// TwinCAT 3 PLC project PLC01
// ProgramVersion: 3.1.4024.0
// libraries:
//   Tc2_Standard, * (Beckhoff Automation GmbH)
//   Tc2_System, * (Beckhoff Automation GmbH)
//   Tc2_Utilities, * (Beckhoff Automation GmbH)
//   Tc3_Module, * (Beckhoff Automation GmbH)
//   VisuDialogs, * (System)
// project tree:
//   DUTs/ st01.TcDUT, st_DirContentInfo.TcDUT
//   / GlobalTextList.TcGTLO, PlcTask.TcTTO, Visualization Manager.TcVMO (not stored), VISU_TASK.TcTTO
//   GVLs/ GVL.TcGVL
//   POUs/ FB_AutoResetBool.TcPOU, FB_FileCopy.TcPOU, MAIN.TcPOU, prgFileHnd.TcPOU, prgFileManipulation.TcPOU
//   VISUs/ Visualization.TcVIS
// real-time tasks:
//   TASK PlcTask: cycle T#10ms, priority 20, ADS port 350
//   TASK VISU_TASK: cycle T#100000us, priority 30, ADS port 351

CONFIGURATION PLC01
    RESOURCE PLC ON TwinCAT3
        TASK PlcTask(INTERVAL := T#10ms, PRIORITY := 20);
        TASK VISU_TASK(INTERVAL := T#100000us, PRIORITY := 30);
        PROGRAM MAIN WITH PlcTask : MAIN;
        PROGRAM VisuElems_Visu_Prg WITH VISU_TASK : VisuElems.Visu_Prg;
    END_RESOURCE
END_CONFIGURATION

// ---- DUTs/st01.TcDUT
TYPE st01 :
STRUCT
	r1:LREAL;
	i1:INT;
	s1:STRING;
	s2:STRING;
	r2:LREAL;
	i2:INT;
END_STRUCT
END_TYPE

// ---- DUTs/st_DirContentInfo.TcDUT
TYPE st_DirContentInfo :
STRUCT
	fileName:T_MaxString;
	dataCriacao:DT;
END_STRUCT
END_TYPE

// ---- GVLs/GVL.TcGVL
{attribute 'qualified_only'}
VAR_GLOBAL
	updateFileList: BOOL;
END_VAR

// ---- POUs/MAIN.TcPOU
PROGRAM MAIN
VAR
	aStructs:ARRAY[1..20] OF st01;
	
END_VAR

prgFileHnd();
prgFileManipulation();

END_PROGRAM

// ---- POUs/prgFileHnd.TcPOU
PROGRAM prgFileHnd
VAR
	bWrite			: BOOL := FALSE;(* Rising edge starts program execution *)
	sNetId			: T_AmsNetId := '';	(* TwinCAT system network address *)
	sFileName		: T_MaxString := 'MyFile';(* CSV destination file path and name *)
	bError			: BOOL;
	nErrId			: UDINT;
	hFile			: UINT		:= 0;(* File handle of the source file *)
	step			: DWORD 	:= 0;

	fbFileOpen	: FB_FileOpen;(* Opens file *)
	fbFileClose	: FB_FileClose;(* Closes file *)
	fbFileWrite	: FB_FileWrite;(* Reads binary data *)	
	trig:R_trig;
	sErr: STRING;
	sMsg: STRING;
	
	//Read
	bRead: BOOL;
	sFileNameRead:T_MaxString;
	bErrorRead:BOOL;
	nErrIdRead:UDINT;
	stepRead:UINT;
	hFileRead:UINT;
	trigRead:R_TRIG;
	
	fbFileOpenRead	: FB_FileOpen;(* Opens file *)
	fbFileCloseRead	: FB_FileClose;(* Closes file *)
	fbFileRead	: FB_FileRead;(* Reads binary data *)
	
	sMsgRead: STRING;
	sErrRead: STRING;
//	sFilePath:T_MaxString:='C:\Relat\';
	sFullfileName: T_MaxString;
END_VAR

trig(CLK:= bWrite);

CASE step OF 
	0:
		IF trig.Q THEN
			step:=10;
			fbFileOpen(bExecute:= FALSE);
			fbFileClose(bExecute:= FALSE);
			fbFileWrite(bExecute:= FALSE);
			sMsg:='Abrindo arquivo';
			sErr:='';
		END_IF
	10:
		sFullfileName:= concat(prgFileManipulation.path, concat(concat('\', sFileName),'.bkp'));
		fbFileOpen(sNetId:=sNetId , sPathName:= sFullfileName, nMode:= FOPEN_MODEWRITE OR FOPEN_MODEBINARY, 
			ePath:= PATH_GENERIC, bExecute:= TRUE, tTimeout:= T#10S, bError => bError, nErrId => nErrId);
		IF NOT fbFileOpen.bBusy THEN
			IF NOT fbFileOpen.bError THEN
				step:=20;
				hFile:= fbFileOpen.hFile;
				sMsg:='Escrevendo arquivo';
			ELSE
				step:=100;
				sErr:='Erro ao abrir o arquivo';
			END_IF
		END_IF
	20:
		fbFileWrite(sNetId:= sNetId, hFile:= hFile,	pWriteBuff:=ADR(main.aStructs), cbWriteLen:= SIZEOF(MAIN.aStructs),
			bExecute:= TRUE,tTimeout:=T#20S, bError => bError, nErrId => nErrId);
		IF NOT fbFileWrite.bBusy THEN
			IF NOT fbFileWrite.bError THEN
				step:=30;
				sMsg:='Arquivo salvo';
			ELSE
				step:=100;
				sErr:='Erro ao escrever o arquivo';	
			END_IF
		END_IF
	30:
		fbFileClose( sNetId := sNetId, hFile := hFile, bExecute := TRUE, bError => bError, nErrId => nErrId);
		IF NOT fbFileClose.bBusy THEN
			step:=100;
			hFile:=0;
			GVL.updateFileList:=TRUE;
		END_IF
	100:
		IF hFile <> 0 THEN
			step:=30;
		ELSE
			step:=0;
			sMsg:='';
		END_IF
END_CASE

trigRead(CLK:= bRead);
CASE stepRead OF
	0:
		IF trigRead.Q THEN
			stepRead:=10;
			fbFileOpenRead(bExecute:= FALSE);
			fbFileCloseRead(bExecute:= FALSE);
			fbFileRead(bExecute:= FALSE);
			sMsgRead:='Abrindo arquivo';
			sErrRead:='';
		END_IF
	10:
		sFileNameRead:= concat(prgFileManipulation.path, concat('\',prgFileManipulation.selectedLocalFile));
		fbFileOpenRead(sNetId:=sNetId , sPathName:= sFileNameRead, nMode:= FOPEN_MODEREAD OR FOPEN_MODEBINARY, 
			ePath:= PATH_GENERIC, bExecute:= TRUE, tTimeout:= T#10S, bError => bErrorRead, nErrId => nErrIdRead);
		IF NOT fbFileOpenRead.bBusy THEN
			IF NOT fbFileOpenRead.bError THEN
				hFileRead:= fbFileOpenRead.hFile;
				stepRead:=20;
			ELSE
				stepRead:=100;	
				sErrRead:='Erro ao abrir arquivo para leitura';
			END_IF
		END_IF
	20:
		fbFileRead(sNetId:=sNetId ,hFile:=hFileRead ,pReadBuff:=ADR(MAIN.aStructs) ,cbReadLen:=SIZEOF(MAIN.aStructs) ,bExecute:=TRUE , 
			tTimeout:= T#30S,bError=> bErrorRead, nErrId=>nErrIdRead);
		IF NOT fbFileRead.bBusy THEN
			IF NOT fbFileRead.bError THEN
				stepRead:=30;
			ELSE
				stepRead:=100;
				sErrRead:='Erro ao ler o arquivo';
			END_IF
		END_IF
	30:
		fbFileCloseRead( sNetId := sNetId, hFile := hFileRead, bExecute := TRUE, bError => bErrorRead, nErrId => nErrIdRead);
		IF NOT fbFileCloseRead.bBusy THEN
			stepRead:=100;
			hFileRead:=0;
			GVL.updateFileList:=TRUE;
		END_IF
	100:
		IF hFileRead <> 0 THEN
			stepRead:=30;
		ELSE
			stepRead:=0;
			sMsgRead:='';
		END_IF
END_CASE

END_PROGRAM

// ---- POUs/prgFileManipulation.TcPOU
PROGRAM prgFileManipulation
VAR
	//Local
	findFiles:FB_EnumFindFileList;
	path: T_MaxString := 'C:\Relat';
	filesFound:ARRAY[1..iNumFiles] OF ST_FindFileEntry;
	filesInfo:ARRAY[1..iNumFiles] OF st_DirContentInfo;
	nNumFiles: UDINT;
	bFindFiles: BOOL;
	bErr: BOOL;
	nErr: UDINT;
	i: UINT;
	i2: UINT;
	searchPath: T_MaxString;
	findFilesFinished:F_TRIG;
	deleteLocalFile: BOOL;

	
	//USB
	findFilesUSB:FB_EnumFindFileList;
	pathUSB: T_MaxString := 'D:';
	filesFoundUSB:ARRAY[1..iNumFiles] OF ST_FindFileEntry;
	filesInfoUSB:ARRAY[1..iNumFiles] OF st_DirContentInfo;
	nNumFilesUSB: UDINT;
	bFindFilesUSB: BOOL;
	bErrUSB: BOOL;
	nErrUSB: UDINT;
	iUSB: UINT;
	i2USB: UINT;
	searchPathUSB: T_MaxString;
	findFilesFinishedUSB:F_TRIG;
	deleteUSBFile: BOOL;

	
	//File copy
	
	fileCopy:FB_FileCopy;
	fileDelete:FB_FileDelete;
	selectedLocalFile:T_MaxString;
	selectedUSBFile:T_MaxString;
	selectedRowLocal:INT;
	selectedRowUSB:INT;
	copyLocalTOUSB: BOOL;
	copyUSBToLocal: BOOL;

	sFullCopyPathLocal: T_MaxString;
	sFullCopyPathUSB: T_MaxString;
	trigCopyLocalUSB, trigCopyUSBLocal, trigDelLocal, trigDelUSB:R_TRIG;
	copyEndTrig, delEndTrig:F_TRIG;
	sCopyMsg: STRING;
	resetUpdateVar:FB_AutoResetBool;
END_VAR
VAR CONSTANT
	iNumFiles:UINT:=10;
END_VAR

searchPath:= concat(path, '\*.*');
findFiles(
	sNetId:='' , 
	sPathName:= searchPath, 
	eCmd:=, 
	pFindList:= ADR(filesFound), 
	cbFindList:= SIZEOF(filesFound), 
	bExecute:= bFindFiles OR GVL.updateFileList, 
	tTimeout:= T#10S, 
	bBusy=> , 
	bError=> bErr, 
	nErrID=> nErr, 
	bEOE=> , 
	nFindFiles=> nNumFiles);

findFilesFinished(CLK:=findFiles.bBusy);

IF findFilesFinished.Q THEN
	FOR i:= 1 TO iNumFiles DO
		filesInfo[i].fileName:= '';
		filesInfo[i].dataCriacao:= DT#1970-1-1-0:0:0;
	END_FOR
	i:=i2:= 1;

	WHILE i<= iNumFiles AND_THEN filesFound[i].sFileName <> '' DO
		IF filesFound[i].fileAttributes.bArchive THEN
			filesInfo[i2].fileName:= filesFound[i].sFileName;
			filesInfo[i2].dataCriacao:= FILETIME_TO_DT(filesFound[i].creationTime);
			i2:=i2+1;
		END_IF
		i:=i+1;
	END_WHILE
END_IF

//USB
searchPathUSB:= concat(pathUSB, '\*.*');
findFilesUSB(
	sNetId:='' , 
	sPathName:= searchPathUSB, 
	eCmd:=, 
	pFindList:= ADR(filesFoundUSB), 
	cbFindList:= SIZEOF(filesFoundUSB), 
	bExecute:= bFindFilesUSB OR GVL.updateFileList, 
	tTimeout:= T#10S, 
	bBusy=> , 
	bError=> bErrUSB, 
	nErrID=> nErrUSB, 
	bEOE=> , 
	nFindFiles=> nNumFilesUSB);

findFilesFinishedUSB(CLK:=findFilesUSB.bBusy);	

IF findFilesFinishedUSB.Q THEN
	
	FOR i:=1 TO iNumFiles DO
		filesInfoUSB[i].fileName:='';
		filesInfoUSB[i].dataCriacao:= DT#1970-1-1-0:0:0;
	END_FOR
	iUSB:=i2USB:= 1;
    
    WHILE iUSB<= iNumFiles AND_THEN filesFoundUSB[iUSB].sFileName <> '' DO
    	IF filesFoundUSB[iUSB].fileAttributes.bArchive THEN
    		filesInfoUSB[i2USB].fileName:= filesFoundUSB[iUSB].sFileName;
    		filesInfoUSB[i2USB].dataCriacao:= FILETIME_TO_DT(filesFoundUSB[iUSB].creationTime);
    		i2USB:=i2USB+1;
    	END_IF
    	iUSB:=iUSB+1;
    END_WHILE
END_IF

IF selectedRowLocal>= 1 AND selectedRowLocal <= iNumFiles THEN
	selectedLocalFile:=filesInfo[selectedRowLocal].fileName;
END_IF	
IF selectedRowUSB>= 1 AND selectedRowUSB <= iNumFiles THEN
	selectedUSBFile:=filesInfoUSB[selectedRowUSB].fileName;
END_IF	

sFullCopyPathLocal:= concat(path,concat('\',selectedLocalFile));
sFullCopyPathUSB:= concat(pathUSB,concat('\',selectedUSBFile));

trigCopyLocalUSB(CLK:= copyLocalTOUSB);
trigCopyUSBLocal(CLK:= copyUSBToLocal);
trigDelLocal(CLK:= deleteLocalFile);
trigDelUSB(CLK:= deleteUSBFile);

IF trigCopyLocalUSB.Q THEN
	fileCopy.sSrcPathName:=sFullCopyPathLocal;
	fileCopy.sDestPathName:= concat(pathUSB,concat('\',selectedLocalFile));
ELSIF trigCopyUSBLocal.Q THEN
	fileCopy.sSrcPathName:=sFullCopyPathUSB;
	fileCopy.sDestPathName:= concat(path,concat('\',selectedUSBFile));;	
END_IF

fileCopy(
	sSrcNetId:= '', 
	sDestNetId:= '', 
	bExecute:=trigCopyLocalUSB.Q OR trigCopyUSBLocal.Q , 
	tTimeOut:= T#20S, 
	bBusy=> , 
	bError=> , 
	nErrId=> );
	
copyEndTrig(CLK:=fileCopy.bBusy);
IF copyEndTrig.Q THEN
	IF NOT fileCopy.bError THEN
		sCopyMsg:='Arquivo copiado com sucesso';
	ELSE 
		sCopyMsg:= concat('Erro na copia do arquivo : ', UDINT_TO_STRING(fileCopy.nErrId));
	END_IF
	GVL.updateFileList:=TRUE;
END_IF



IF trigDelLocal.Q THEN
	fileDelete.sPathName:= sFullCopyPathLocal;
ELSIF trigDelUSB.Q THEN
	fileDelete.sPathName:= sFullCopyPathUSB;	
END_IF

fileDelete(
	sNetId:= '', 
	sPathName:= , 
	ePath:= , 
	bExecute:= trigDelLocal.Q OR trigDelUSB.Q , 
	tTimeout:= T#20S, 
	bBusy=> , 
	bError=> , 
	nErrId=> );
	
delEndTrig(CLK:= fileDelete.bBusy);
IF delEndTrig.Q THEN
	GVL.updateFileList:=TRUE;
END_IF

//put this on the last line
resetUpdateVar(tResetTime:=T#100MS , bReset:= GVL.updateFileList);

END_PROGRAM

// ---- POUs/FB_FileCopy.TcPOU
FUNCTION_BLOCK FB_FileCopy
VAR_INPUT
	sSrcNetId			: T_AmsNetId;	(* TwinCAT network address of the source file *)
	sSrcPathName		: T_MaxString;	(* Source file path and name *)
	sDestNetId			: T_AmsNetId;	(* TwinCAT network address of the destination file *)
	sDestPathName		: T_MaxString;  (* Destination file path and name *)
	bExecute			: BOOL;			(* Rising edge start fb execution *)
	tTimeOut			: TIME := DEFAULT_ADS_TIMEOUT;(* Max. ADS timeout time *)
END_VAR
VAR_OUTPUT
	bBusy				:BOOL;(* TRUE => File copy execution in progress, FALSE => File copy execution idle *)
	bError				:BOOL;(* TRUE => Error, FALSE => No error *)
	nErrId				:UDINT;(* Error code *)
END_VAR
VAR
	fbFileOpen			:FB_FileOpen;
	fbFileClose			:FB_FileClose;
	fbFileRead			:FB_FileRead;
	fbFileWrite			:FB_FileWrite;

	hSrcFile				:UINT	:= 0;(* File handle of the source file *)
	hDestFile			:UINT	:= 0;(* File handle of the destination file *)

	Step				:DWORD;
	RisingEdge			:R_TRIG;

	buffRead				:ARRAY[1..1000] OF BYTE;(* Buffer *)
	cbReadLength		:UDINT := 0;
END_VAR

RisingEdge(CLK:=bExecute);

CASE Step OF
	0:	(* Idle state *)
		IF RisingEdge.Q THEN
			bBusy := TRUE;
			bError:= FALSE;
			nErrId:=0;
			Step := 1;
			cbReadLength:=0;
			hSrcFile:=0;
			hDestFile:=0;
		END_IF

	1:	(* Open source file *)
		fbFileOpen( bExecute := FALSE );
		fbFileOpen( sNetId := sSrcNetId, sPathName := sSrcPathName,
					nMode := FOPEN_MODEREAD OR FOPEN_MODEBINARY,
					ePath := PATH_GENERIC, tTimeout := tTimeOut, bExecute := TRUE );
		Step := Step + 1;
	2:
		fbFileOpen( bExecute := FALSE );
		IF NOT fbFileOpen.bBusy THEN
			IF fbFileOpen.bError THEN
				nErrId := fbFileOpen.nErrId;
				bError := TRUE;
				Step := 50;
			ELSE
				hSrcFile := fbFileOpen.hFile;
				Step := Step + 1;
			END_IF
		END_IF

	3:	(* Open destination file *)
		fbFileOpen( bExecute := FALSE );
		fbFileOpen( sNetId := sDestNetId, sPathName := sDestPathName,
					nMode := FOPEN_MODEWRITE OR FOPEN_MODEBINARY,
					ePath := PATH_GENERIC, tTimeout := tTimeOut, bExecute := TRUE );
		Step := Step+1;
	4:
		fbFileOpen( bExecute := FALSE );
		IF NOT fbFileOpen.bBusy THEN
			IF fbFileOpen.bError THEN
				nErrId := fbFileOpen.nErrId;
				bError := TRUE;
				Step := 50;
			ELSE
				hDestFile := fbFileOpen.hFile;
				Step := Step + 1;
			END_IF
		END_IF

	5:	(* Read data from source file *)
		cbReadLength := 0;
		fbFileRead( bExecute:= FALSE );
		fbFileRead( sNetId:=sSrcNetId, hFile:=hSrcFile,
					pReadBuff:= ADR(buffRead), cbReadLen:= SIZEOF(buffRead),
					bExecute:=TRUE, tTimeout:=tTimeOut );
		Step := Step + 1;
	6:
		fbFileRead( bExecute:= FALSE );
		IF NOT fbFileRead.bBusy THEN
			IF fbFileRead.bError THEN
				nErrId := fbFileRead.nErrId;
				bError := TRUE;
				Step := 50;
			ELSE
				cbReadLength := fbFileRead.cbRead;
				Step := Step + 1;
			END_IF
		END_IF

	7:	(* Write data to destination file *)
		fbFileWrite( bExecute := FALSE );
		fbFileWrite( sNetId:=sDestNetId, hFile:=hDestFile,
					pWriteBuff:= ADR(buffRead), cbWriteLen:= cbReadLength,
					bExecute:=TRUE, tTimeout:=tTimeOut );
		Step := Step + 1;
	8:
		fbFileWrite( bExecute := FALSE );
		IF NOT fbFileWrite.bBusy THEN
			IF fbFileWrite.bError THEN
				nErrId := fbFileWrite.nErrId;
				bError := TRUE;
				Step := 50;
			ELSE
				IF fbFileRead.bEOF THEN (* Check if the EOF flag ist set *)
					Step := 50;	(* Cleanup: close the destination and source files *)
				ELSE
					Step := 5; (* Repeat reading/writing *)
				END_IF
			END_IF
		END_IF

	30:	(* Close the destination file *)
		fbFileClose( bExecute := FALSE );
		fbFileClose( sNetId:=sDestNetId, hFile:=hDestFile, bExecute:=TRUE, tTimeout:=tTimeOut );
		Step := Step + 1;
	31:
		fbFileClose( bExecute := FALSE );
		IF NOT fbFileClose.bBusy THEN
			IF fbFileClose.bError THEN
				nErrId := fbFileClose.nErrId;
				bError := TRUE;
			END_IF
			Step := 50;
			hDestFile := 0;
		END_IF

	40: (* Close source file *)
		fbFileClose( bExecute := FALSE );
		fbFileClose( sNetId:=sSrcNetId, hFile:=hSrcFile, bExecute:=TRUE, tTimeout:=tTimeOut );
		Step := Step + 1;
	41:
		fbFileClose( bExecute := FALSE );
		IF NOT fbFileClose.bBusy THEN
			IF fbFileClose.bError THEN
				nErrId := fbFileClose.nErrId;
				bError := TRUE;
			END_IF
			Step := 50;
			hSrcFile := 0;
		END_IF

	50: (* Error or ready => Cleanup *)
		IF ( hDestFile <> 0 ) THEN
			Step := 30; (* Close the destination file*)
		ELSIF (hSrcFile <> 0 ) THEN
			Step := 40; (* Close the source file *)
		ELSE
			Step := 0;	(* Ready *)
			bBusy := FALSE;
		END_IF

END_CASE

END_FUNCTION_BLOCK

// ---- POUs/FB_AutoResetBool.TcPOU
FUNCTION_BLOCK FB_AutoResetBool
VAR_INPUT
	tResetTime:TIME:=T#100MS;
END_VAR
VAR_OUTPUT
END_VAR
VAR
	t1:TON;
END_VAR
VAR_IN_OUT
	bReset: BOOL;
END_VAR

t1(IN:=bReset , PT:= tResetTime);
IF t1.Q THEN
	bReset:=FALSE;
END_IF

END_FUNCTION_BLOCK

// ---- GlobalTextList.TcGTLO
TEXTLIST GlobalTextList
  607 = '%s'
  576 = '<<< Copiar'
  915 = 'Arquivos'
  449 = 'Carregar'
  770 = 'Copiar >>>'
  642 = 'Criação'
  294 = 'Delete'
  875 = 'Destino'
  166 = 'i1'
  223 = 'i2'
  765 = 'Local'
  253 = 'Mensagem : %s'
  932 = 'Nome'
  814 = 'Nome arquivo'
  762 = 'Origem'
  370 = 'r1'
  76 = 'r2'
  950 = 'Refresh'
  338 = 's1'
  862 = 's2'
  813 = 'Salvar'
  575 = 'USB'
END_TEXTLIST

// ---- VISUs/Visualization.TcVIS
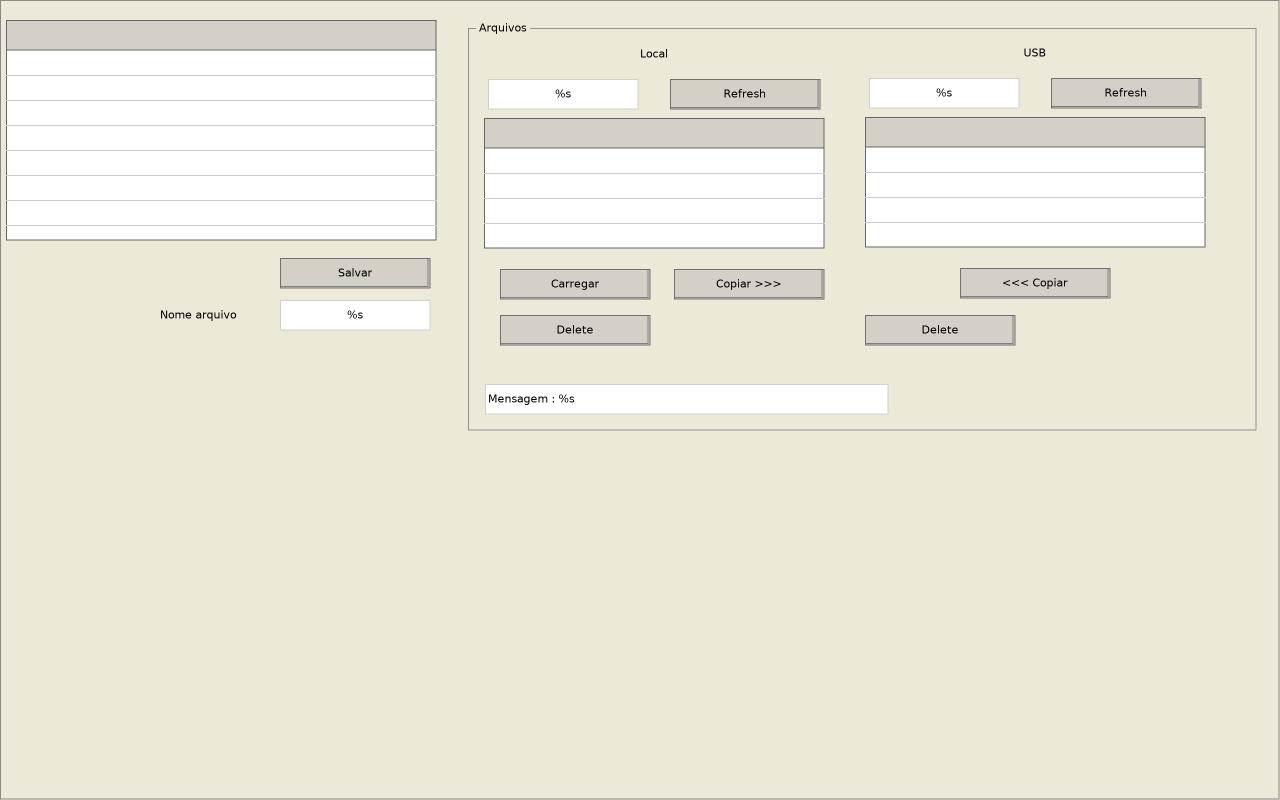
VISUALIZATION Visualization  // 1280x800
    Table (6,20 430x220), data array: MAIN.aStructs
        p3854506369: MAIN.aStructs[INDEX].r1
        p1892666644: MAIN.aStructs[INDEX].i1
        p338671338: MAIN.aStructs[INDEX].s1
        p2170511999: MAIN.aStructs[INDEX].s2
        p3723444502: MAIN.aStructs[INDEX].r2
        p1218418051: MAIN.aStructs[INDEX].i2
    Button (280,258 150x30), "Salvar"
        tap prgFileHnd.bWrite
    Label (144,300 109x30), "Nome arquivo"
    Textfield (280,300 150x30), "%s", text variable: prgFileHnd.sFileName
        OnMouseClick: write the text variable via Default
    GroupBox (468,20 788x410), "Arquivos"
        Table (16,98 340x130), data array: prgFileManipulation.filesInfo
            p3854506369: prgFileManipulation.filesInfo[INDEX].fileName
            p1892666644: prgFileManipulation.filesInfo[INDEX].dataCriacao
            p2232123230: Nome
            p511219082: Criação
            p1137915858: prgFileManipulation.selectedRowLocal
        Textfield (20,59 150x30), "%s", text variable: prgFileManipulation.path
            OnMouseClick: write the text variable via Default
        Button (202,59 150x30), "Refresh"
            tap prgFileManipulation.bFindFiles
        Label (111,19 150x30), "Local"
        Table (397,97 340x130), data array: prgFileManipulation.filesInfoUSB
            p3854506369: prgFileManipulation.filesInfoUSB[INDEX].fileName
            p1892666644: prgFileManipulation.filesInfoUSB[INDEX].dataCriacao
            p2232123230: Nome
            p511219082: Criação
            p1137915858: prgFileManipulation.selectedRowUSB
        Button (206,249 150x30), "Copiar >>>"
            tap prgFileManipulation.copyLocalTOUSB
        Button (492,248 150x30), "<<< Copiar"
            tap prgFileManipulation.copyUSBToLocal
        Textfield (17,364 403x30), "Mensagem : %s", text variable: prgFileManipulation.sCopyMsg
        Button (32,249 150x30), "Carregar"
            tap prgFileHnd.bRead
        Button (32,295 150x30), "Delete"
            tap prgFileManipulation.deleteLocalFile
        Button (397,295 150x30), "Delete"
            tap prgFileManipulation.deleteUSBFile
    Textfield (869,78 150x30), "%s", text variable: prgFileManipulation.pathUSB
        OnMouseClick: write the text variable via Default
    Button (1051,78 150x30), "Refresh"
        tap prgFileManipulation.bFindFilesUSB
    Label (960,38 150x30), "USB"
END_VISUALIZATION
